PROGRAM P_Demo_PTOD_TO_TOD
VAR
    todRealValue           : TOD := TOD#12:34:56; // 模拟 wire 缓冲区中的 TOD 字段
    pTODField              : POINTER TO TOD; // 业务侧先算好的字段地址（ADR 或 pBase+nOff）
    bExtractField          : BOOL; // 在线置 TRUE 触发一次解析
    todRealValue_extracted : TOD; // 解析后的副本，供业务逻辑使用
END_VAR

// ============================================================
// Tc2_Utilities.PTOD_TO_TOD 演示程序（FUNCTION）
// ============================================================
// 场景：从一段二进制 wire 缓冲区里按偏移取 TOD 字段（Modbus/CAN/ADS Raw）。
// 价值：替代手写 pField + nOff + ^ 指针算术；一次调用取值，少打错符号。
// 验证：在线写 todRealValue := TOD#12:34:56；bExtractField := TRUE；
//       下一周期 todRealValue_extracted 应等于 todRealValue。
// ============================================================

// 业务代码通常已经算好字段地址（pBase + 协议偏移）；演示用 ADR 等价
pTODField := ADR(todRealValue);

IF bExtractField AND pTODField <> 0 THEN
    // 单次完整调用：避免手写 ^ 解引用，统一风格便于和字节序转换串联
    todRealValue_extracted := PTOD_TO_TOD(pTODField);
    bExtractField := FALSE;
END_IF;

END_PROGRAM

(* stored: Version 1.1.0.1, ProductVersion 3.1.4024.5
   POU P_Demo_PTOD_TO_TOD: Id {e06867e2-8e3b-5c4d-9872-7bc546ff867d}, SpecialFunc None *)
